FUNCTION_BLOCK FeedReactorLogic (* CAT Function Block Type *)
  (* Standard: 61499-2 *)
  (* Version 1.0, 10/1/2026, Claude/Hidryco, Schneider Electric, Rev1 - Caminho de 3 bombas reescrito (FeedReactor3PsBasic Rev1): mesmo funcionamento da Water Discharge; PID unico (PIDISc.RunPID1/Setpoint1); velocidade unica via SpeedGate (reenvio 1 s); rodizio por horimetro (FB_OPD); velocidade real (FB_SPEED); pH/condutividade pelos alarmes L/H (narrativa); reatores recebem disponibilidade/rodando de qualquer bomba; removidos SpeedSp1-3, InfluentCofiguration, INT2BOOL e WaitingTime (caminho de 1 bomba nao usado) *)
  PACKAGE SE.Nereda;
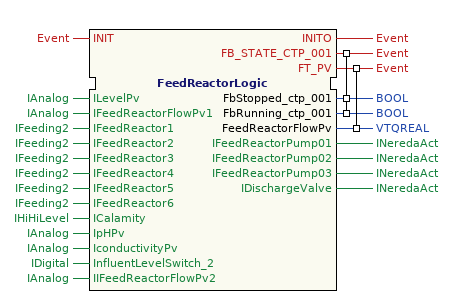
  EVENT_INPUT
    INIT;
  END_EVENT
  EVENT_OUTPUT
    INITO;
    FB_STATE_CTP_001 WITH FbStopped_ctp_001, FbRunning_ctp_001;
    FT_PV WITH FeedReactorFlowPv; (* Request for new value and limits *)
  END_EVENT
  VAR_OUTPUT
    FbStopped_ctp_001 : BOOL;
    FbRunning_ctp_001 : BOOL;
    FeedReactorFlowPv : VTQREAL; (* Vtq value *)
  END_VAR
  SOCKETS
    ILevelPv : IAnalog;
    IFeedReactorFlowPv1 : IAnalog;
    IFeedReactor1 : IFeeding2;
    IFeedReactor2 : IFeeding2;
    IFeedReactor3 : IFeeding2;
    IFeedReactor4 : IFeeding2;
    IFeedReactor5 : IFeeding2;
    IFeedReactor6 : IFeeding2;
    ICalamity : IHiHiLevel;
    IpHPv : IAnalog;
    IconductivityPv : IAnalog;
    InfluentLevelSwitch_2 : IDigital;
  END_SOCKETS
  SOCKETS
    IIFeedReactorFlowPv2 : IAnalog; (* Process value (range considered) interface adapter *)
  END_SOCKETS
  PLUGS
    IFeedReactorPump01 : INeredaAct;
    IFeedReactorPump02 : INeredaAct;
    IFeedReactorPump03 : INeredaAct;
    IDischargeValve : INeredaAct;
  END_PLUGS
  (* 01 - FUNCTIONNAL INPUT INTERFACE *)
  (* 00 - INITIALIZATION *)
  (* 05 - LOGIC *)
  (* 06 - HMI INTERFACE *)
  (* 03 - FIELD INTERFACE *)
  (* Feed Reactor Logic (One Pump) *)
  (* 02 - FUNCTIONNAL OUTPUT INTERFACE *)
  (* Interlock *)
  (* Feed Reactor Logic (3 Pumps) *)
  (* Capacity Setpoint *)
  (* Stop Pumps Cdts : The feed to the reactor must be stopped in the following situations: • Low Low level influent buffer; • pH value influent buffer too low or too high; • conductivity influent buffer too low or too high. *)
  FBS
    IThis : FeedReactorLogic_HMI(QI := TRUE);
    FeedReactorFlowPv_Status : decodeStatus; {SET_ATTRIBUTE(Configuration.Component.HideUnusedPorts, )}
    CmdPumpSmooth : boolValueChanged;
    CmdValveSmooth : boolValueChanged;
    PID : PID;
    LowLowFlow_ctp001 : ilckCondItem(CondCause := Active1);
    LowLowFlowAlarm : AND_88A3DD8EC65DD11C; {SET_ATTRIBUTE(Configuration.GenericFBType.InterfaceParams, Runtime.Standard#CNT:=2;OUT:BOOL)}
    FeedReactor1PLogic : FeedReactor1PBasic;
    LevelPv_Status : decodeStatus;
    ForceStopPump : OR_88A3DD8EC65DD11C(IN1 := FALSE); {SET_ATTRIBUTE(Configuration.GenericFBType.InterfaceParams, Runtime.Standard#CNT:=2;OUT:BOOL)}
    RESET_BTNs : RESET_BTNs;
    LoLoFlowAlarmManager : DelayedActive(pin_4E076A4928A0DFEF := TRUE, pin_1CE054BDD0AD4DEB := T#1m);
    HighHighLevel_Calamity : ilckCondItem(CondCause := Active1);
    HighHighCalamity : OR_88A3DD8EC65DD11C; {SET_ATTRIBUTE(Configuration.GenericFBType.InterfaceParams, Runtime.Standard#CNT:=2;OUT:BOOL)}
    CmdPump : BOOL2INT;
    CmdValve : BOOL2INT;
    ResetReq : OR_1147623A96AA66A8; {SET_ATTRIBUTE(Configuration.GenericFBType.InterfaceParams, Runtime.Standard#CNT:=7;OUT:BOOL)}
    FeedPumpFbMng : FeedPumpFbReactor;
    FeedReactor3PsLogic : FeedReactor3PsBasic; {SET_ATTRIBUTE(Configuration.Component.HideUnusedPorts, )}
    CmdPump1Smooth : boolValueChanged;
    CmdPump2Smooth : boolValueChanged;
    CmdPump1 : BOOL2INT;
    CmdPump2 : BOOL2INT;
    CmdPump3Smooth : boolValueChanged;
    CmdPump3 : BOOL2INT;
    ForceStop : OR_169B00D031196E7C4; {SET_ATTRIBUTE(Configuration.GenericFBType.InterfaceParams, Runtime.Standard#CNT:=4;OUT:BOOL)}
    pH_Status : decodeStatus; {SET_ATTRIBUTE(Configuration.Component.HideUnusedPorts, )}
    conductivity_Status : decodeStatus; {SET_ATTRIBUTE(Configuration.Component.HideUnusedPorts, )}
    PIDISc : PID3_Manager;
    OR1 : OR_550FE6D62F509EB3; {SET_ATTRIBUTE(Configuration.GenericFBType.InterfaceParams, Runtime.Standard#CNT:=3;OUT:BOOL)}
    INT2BOOL1 : INT2BOOL;
    TickCycle : E_CYCLE(DT := T#1s);
    SpeedGate : E_PERMIT;
    Autotune1 : Autotune;
  END_FBS
  EVENT_CONNECTIONS
    LowLowFlowAlarm.CNF TO LowLowFlow_ctp001.REQ;
    IFeedReactorFlowPv1.REQ_STATUS TO FeedReactorFlowPv_Status.REQ;
    FeedReactorFlowPv_Status.CNF TO LowLowFlowAlarm.REQ;
    ILevelPv.REQ_STATUS TO LevelPv_Status.REQ;
    LowLowFlowAlarm.CNF TO ForceStopPump.REQ;
    OR1.CNF TO ForceStopPump.REQ;
    INIT TO IThis.DA969393F6D27920;
    IThis.A8EF0BC2917800E0 TO IThis.3D88186A4172EAF0;
    HighHighCalamity.CNF TO HighHighLevel_Calamity.REQ;
    FeedReactor1PLogic.078EA09CED294ADE TO IThis.ACDDFE951F9AC365;
    RESET_BTNs.920962203CA54948 TO IThis.B1F8118D15146EFE;
    IThis.25C5B7DA6CF97B41 TO FeedReactor1PLogic.A69A10F93A67179B;
    IThis.25C5B7DA6CF97B41 TO RESET_BTNs.AB695E9A35A20E19;
    IThis.67B3DB0A1F2CCD1E TO RESET_BTNs.AB695E9A35A20E19;
    OR1.CNF TO IFeedReactor1.5A11906EF1EE87B0;
    OR1.CNF TO IFeedReactor2.5A11906EF1EE87B0;
    OR1.CNF TO IFeedReactor3.5A11906EF1EE87B0;
    OR1.CNF TO IFeedReactor4.5A11906EF1EE87B0;
    OR1.CNF TO IFeedReactor5.5A11906EF1EE87B0;
    OR1.CNF TO IFeedReactor6.5A11906EF1EE87B0;
    OR1.CNF TO CmdPump.DD5870AA881150BB;
    IFeedReactorFlowPv1.REQ TO IFeedReactor1.7593DE3331C575B6;
    IFeedReactorFlowPv1.REQ TO IFeedReactor2.7593DE3331C575B6;
    IFeedReactorFlowPv1.REQ TO IFeedReactor3.7593DE3331C575B6;
    IFeedReactorFlowPv1.REQ TO IFeedReactor4.7593DE3331C575B6;
    IFeedReactorFlowPv1.REQ TO IFeedReactor5.7593DE3331C575B6;
    IFeedReactorFlowPv1.REQ TO IFeedReactor6.7593DE3331C575B6;
    IFeedReactorPump01.CC753684FA882790 TO IFeedReactor3.70EEE9F2AA8AC204;
    IFeedReactorPump01.CC753684FA882790 TO IFeedReactor4.70EEE9F2AA8AC204;
    IFeedReactorPump01.CC753684FA882790 TO IFeedReactor5.70EEE9F2AA8AC204;
    IFeedReactorPump01.CC753684FA882790 TO IFeedReactor6.70EEE9F2AA8AC204;
    IFeedReactor1.74BA0DB8212F2576 TO FeedReactor1PLogic.7E30127865CFE16B;
    IFeedReactor2.74BA0DB8212F2576 TO FeedReactor1PLogic.7E30127865CFE16B;
    IFeedReactor3.74BA0DB8212F2576 TO FeedReactor1PLogic.7E30127865CFE16B;
    IFeedReactor4.74BA0DB8212F2576 TO FeedReactor1PLogic.7E30127865CFE16B;
    IFeedReactor5.74BA0DB8212F2576 TO FeedReactor1PLogic.7E30127865CFE16B;
    IFeedReactor6.74BA0DB8212F2576 TO FeedReactor1PLogic.7E30127865CFE16B;
    IFeedReactor1.8D6216DA6F1D1AB3 TO FeedReactor1PLogic.595E94AC272AAE70;
    IFeedReactor2.8D6216DA6F1D1AB3 TO FeedReactor1PLogic.595E94AC272AAE70;
    IFeedReactor3.8D6216DA6F1D1AB3 TO FeedReactor1PLogic.595E94AC272AAE70;
    IFeedReactor4.8D6216DA6F1D1AB3 TO FeedReactor1PLogic.595E94AC272AAE70;
    IFeedReactor5.8D6216DA6F1D1AB3 TO FeedReactor1PLogic.595E94AC272AAE70;
    IFeedReactor6.8D6216DA6F1D1AB3 TO FeedReactor1PLogic.595E94AC272AAE70;
    IDischargeValve.9CD053F8408797ED TO FeedReactor1PLogic.FBAC3AB0F3E1774A;
    IFeedReactorPump01.9CD053F8408797ED TO FeedReactor1PLogic.8666C65DB2F34DF4;
    IFeedReactorPump01.CC753684FA882790 TO FeedReactor1PLogic.01DE5B3982687378;
    IDischargeValve.CC753684FA882790 TO FeedReactor1PLogic.EBB538FC7819A0F0;
    ForceStopPump.CNF TO FeedReactor1PLogic.4BDCB67B4FFE0D64;
    FeedReactor1PLogic.085A47BAE233EC43 TO CmdPumpSmooth.REQ;
    FeedReactor1PLogic.BA495A2CD6F37AAA TO CmdValveSmooth.REQ;
    CmdPumpSmooth.CHD TO CmdPump.DD5870AA881150BB;
    CmdValveSmooth.CHD TO CmdValve.DD5870AA881150BB;
    IThis.A8EF0BC2917800E0 TO PIDISc.INIT;
    PIDISc.CE80458C9D5EF15A TO INITO;
    LoLoFlowAlarmManager.DDA64CDC00519DA4 TO LowLowFlowAlarm.REQ;
    ICalamity.15126F43E529BB4F TO HighHighCalamity.REQ;
    CmdValve.6FC99A5BD1C38561 TO IDischargeValve.0F1CDF9A9B4A227A;
    IFeedReactorPump01.9CD053F8408797ED TO FB_STATE_CTP_001;
    IFeedReactorFlowPv1.REQ TO FT_PV;
    IThis.67B3DB0A1F2CCD1E TO ResetReq.REQ;
    IFeedReactorPump01.9CD053F8408797ED TO ResetReq.REQ;
    ResetReq.CNF TO LoLoFlowAlarmManager.C451626F7187F42D;
    IFeedReactor2.9C2DC160D0649F17 TO ResetReq.REQ;
    IFeedReactor1.9C2DC160D0649F17 TO ResetReq.REQ;
    IFeedReactor3.9C2DC160D0649F17 TO ResetReq.REQ;
    IFeedReactor4.9C2DC160D0649F17 TO ResetReq.REQ;
    IFeedReactor5.9C2DC160D0649F17 TO ResetReq.REQ;
    IFeedReactor6.9C2DC160D0649F17 TO ResetReq.REQ;
    FeedPumpFbMng.CC5621380E74A0E0 TO IFeedReactor1.03923062E780DBFC;
    FeedPumpFbMng.CC5621380E74A0E0 TO IFeedReactor2.03923062E780DBFC;
    FeedPumpFbMng.CC5621380E74A0E0 TO IFeedReactor3.03923062E780DBFC;
    FeedPumpFbMng.CC5621380E74A0E0 TO IFeedReactor4.03923062E780DBFC;
    FeedPumpFbMng.CC5621380E74A0E0 TO IFeedReactor5.03923062E780DBFC;
    FeedPumpFbMng.CC5621380E74A0E0 TO IFeedReactor6.03923062E780DBFC;
    IFeedReactor1.64A31C18B824409C TO FeedPumpFbMng.84006066E90F70DE;
    IFeedReactor2.64A31C18B824409C TO FeedPumpFbMng.84006066E90F70DE;
    IFeedReactor3.64A31C18B824409C TO FeedPumpFbMng.84006066E90F70DE;
    IFeedReactor4.64A31C18B824409C TO FeedPumpFbMng.84006066E90F70DE;
    IFeedReactor5.64A31C18B824409C TO FeedPumpFbMng.84006066E90F70DE;
    IFeedReactor6.64A31C18B824409C TO FeedPumpFbMng.84006066E90F70DE;
    IFeedReactor1.74BA0DB8212F2576 TO FeedReactor1PLogic.595E94AC272AAE70;
    IFeedReactor2.74BA0DB8212F2576 TO FeedReactor1PLogic.595E94AC272AAE70;
    IFeedReactor3.74BA0DB8212F2576 TO FeedReactor1PLogic.595E94AC272AAE70;
    IFeedReactor4.74BA0DB8212F2576 TO FeedReactor1PLogic.595E94AC272AAE70;
    IFeedReactor5.74BA0DB8212F2576 TO FeedReactor1PLogic.595E94AC272AAE70;
    IFeedReactor6.74BA0DB8212F2576 TO FeedReactor1PLogic.595E94AC272AAE70;
    CmdPump1Smooth.CHD TO CmdPump1.DD5870AA881150BB;
    CmdPump2Smooth.CHD TO CmdPump2.DD5870AA881150BB;
    CmdPump3Smooth.CHD TO CmdPump3.DD5870AA881150BB;
    CmdPump1Smooth.CNF TO CmdPump2Smooth.REQ;
    CmdPump2Smooth.CNF TO CmdPump3Smooth.REQ;
    CmdPump2.6FC99A5BD1C38561 TO IFeedReactorPump02.0F1CDF9A9B4A227A;
    CmdPump3.6FC99A5BD1C38561 TO IFeedReactorPump03.0F1CDF9A9B4A227A;
    IpHPv.REQ_STATUS TO pH_Status.REQ;
    IconductivityPv.REQ_STATUS TO conductivity_Status.REQ;
    OR1.CNF TO ForceStop.REQ;
    pH_Status.CNF TO ForceStop.REQ;
    conductivity_Status.CNF TO ForceStop.REQ;
    InfluentLevelSwitch_2.REQ TO INT2BOOL1.DD5870AA881150BB;
    INT2BOOL1.6FC99A5BD1C38561 TO OR1.REQ;
    LevelPv_Status.CNF TO OR1.REQ;
    IThis.A8EF0BC2917800E0 TO TickCycle.START;
    TickCycle.EO TO FeedReactor3PsLogic.471C3CADA717EC13;
    TickCycle.EO TO SpeedGate.EI;
    FeedReactor3PsLogic.54C5C4335FC174B1 TO SpeedGate.EI;
    SpeedGate.EO TO IFeedReactorPump01.1E00729184986247;
    IFeedReactorPump01.9CD053F8408797ED TO FeedReactor3PsLogic.8666C65DB2F34DF4;
    IFeedReactorPump01.CC753684FA882790 TO FeedReactor3PsLogic.01DE5B3982687378;
    IFeedReactorPump01.2DA8AEC15204E92D TO FeedReactor3PsLogic.168409FF111F0B5A;
    IFeedReactorPump01.F846995A4121D865 TO FeedReactor3PsLogic.5E41A10D869921BD;
    SpeedGate.EO TO IFeedReactorPump02.1E00729184986247;
    IFeedReactorPump02.9CD053F8408797ED TO FeedReactor3PsLogic.8666C65DB2F34DF4;
    IFeedReactorPump02.CC753684FA882790 TO FeedReactor3PsLogic.01DE5B3982687378;
    IFeedReactorPump02.2DA8AEC15204E92D TO FeedReactor3PsLogic.168409FF111F0B5A;
    IFeedReactorPump02.F846995A4121D865 TO FeedReactor3PsLogic.5E41A10D869921BD;
    SpeedGate.EO TO IFeedReactorPump03.1E00729184986247;
    IFeedReactorPump03.9CD053F8408797ED TO FeedReactor3PsLogic.8666C65DB2F34DF4;
    IFeedReactorPump03.CC753684FA882790 TO FeedReactor3PsLogic.01DE5B3982687378;
    IFeedReactorPump03.2DA8AEC15204E92D TO FeedReactor3PsLogic.168409FF111F0B5A;
    IFeedReactorPump03.F846995A4121D865 TO FeedReactor3PsLogic.5E41A10D869921BD;
    FeedReactor3PsLogic.085A47BAE233EC43 TO CmdPump1Smooth.REQ;
    CmdPump1.6FC99A5BD1C38561 TO IFeedReactorPump01.0F1CDF9A9B4A227A;
    IFeedReactor1.74BA0DB8212F2576 TO FeedReactor3PsLogic.7E30127865CFE16B;
    IFeedReactor1.74BA0DB8212F2576 TO FeedReactor3PsLogic.595E94AC272AAE70;
    IFeedReactor1.8D6216DA6F1D1AB3 TO FeedReactor3PsLogic.595E94AC272AAE70;
    FeedReactor3PsLogic.FCD297844523CE03 TO IFeedReactor1.70EEE9F2AA8AC204;
    IFeedReactor2.74BA0DB8212F2576 TO FeedReactor3PsLogic.7E30127865CFE16B;
    IFeedReactor2.74BA0DB8212F2576 TO FeedReactor3PsLogic.595E94AC272AAE70;
    IFeedReactor2.8D6216DA6F1D1AB3 TO FeedReactor3PsLogic.595E94AC272AAE70;
    FeedReactor3PsLogic.FCD297844523CE03 TO IFeedReactor2.70EEE9F2AA8AC204;
    FeedReactor3PsLogic.FCD297844523CE03 TO FeedPumpFbMng.84006066E90F70DE;
    ForceStop.CNF TO FeedReactor3PsLogic.4BDCB67B4FFE0D64;
    LevelPv_Status.CNF TO FeedReactor3PsLogic.4BDCB67B4FFE0D64;
    FeedReactorFlowPv_Status.CNF TO FeedReactor3PsLogic.16643588834996DE;
    IFeedReactorFlowPv1.REQ TO FeedReactor3PsLogic.16643588834996DE;
    PID.CNF TO FeedReactor3PsLogic.0510D36B485733F5;
    FeedReactor3PsLogic.1878369CED9D9897 TO PIDISc.REQ;
    IThis.B4CA49BBBE66E908 TO FeedReactor3PsLogic.6712A6C827380130;
    IThis.C0050F7CE802CE26 TO FeedReactor3PsLogic.6712A6C827380130;
    IThis.25C5B7DA6CF97B41 TO FeedReactor3PsLogic.A69A10F93A67179B;
    FeedReactor3PsLogic.50ABF706162D6E5D TO IThis.E675E5B2A8A39442;
  END_CONNECTIONS
  DATA_CONNECTIONS
    LowLowFlowAlarm.OUT TO LowLowFlow_ctp001.CondSignal;
    IFeedReactorFlowPv1.Status TO FeedReactorFlowPv_Status.Status;
    FeedReactorFlowPv_Status.LoLoAlarm TO LowLowFlowAlarm.IN2;
    ILevelPv.Status TO LevelPv_Status.Status;
    LevelPv_Status.LoLoAlarm TO ForceStopPump.IN2;
    HighHighCalamity.OUT TO HighHighLevel_Calamity.CondSignal;
    FeedReactor1PLogic.AE321536059FD861 TO IThis.B8642C11FD7EB72C;
    IThis.F8C15B6A2368EBC2 TO FeedReactor1PLogic.2AC43BA050B74406;
    IThis.F8C15B6A2368EBC2 TO RESET_BTNs.479D4538AEFD6EE1;
    IThis.78DC25A16E3E12D4 TO RESET_BTNs.26767209E3135B52;
    OR1.OUT TO IFeedReactor1.2B9DC646C4F67E84;
    OR1.OUT TO IFeedReactor2.2B9DC646C4F67E84;
    OR1.OUT TO IFeedReactor3.2B9DC646C4F67E84;
    OR1.OUT TO IFeedReactor4.2B9DC646C4F67E84;
    OR1.OUT TO IFeedReactor5.2B9DC646C4F67E84;
    OR1.OUT TO IFeedReactor6.2B9DC646C4F67E84;
    IFeedReactorFlowPv1.Value TO IFeedReactor5.E608EE3E510ADBC9;
    IFeedReactorFlowPv1.Value TO IFeedReactor6.E608EE3E510ADBC9;
    IFeedReactorFlowPv1.Value TO IFeedReactor4.E608EE3E510ADBC9;
    IFeedReactorFlowPv1.Value TO IFeedReactor3.E608EE3E510ADBC9;
    IFeedReactorFlowPv1.Value TO IFeedReactor2.E608EE3E510ADBC9;
    IFeedReactorFlowPv1.Value TO IFeedReactor1.E608EE3E510ADBC9;
    IFeedReactorPump01.8A8A07EFCDA1443C TO IFeedReactor6.B41B0731DC9AD731;
    IFeedReactorPump01.8A8A07EFCDA1443C TO IFeedReactor5.B41B0731DC9AD731;
    IFeedReactorPump01.8A8A07EFCDA1443C TO IFeedReactor4.B41B0731DC9AD731;
    IFeedReactorPump01.8A8A07EFCDA1443C TO IFeedReactor3.B41B0731DC9AD731;
    IFeedReactor1.9A80F414E2AF6B87 TO FeedReactor1PLogic.C915B42A7E29ABA7;
    IFeedReactor2.9A80F414E2AF6B87 TO FeedReactor1PLogic.C035C9DDF73934B1;
    IFeedReactor3.9A80F414E2AF6B87 TO FeedReactor1PLogic.BA46BCD3AD3C4E0E;
    IFeedReactor4.9A80F414E2AF6B87 TO FeedReactor1PLogic.05202F12A8CD5CAE;
    IFeedReactor5.9A80F414E2AF6B87 TO FeedReactor1PLogic.D190D2DBF4763077;
    IFeedReactor6.9A80F414E2AF6B87 TO FeedReactor1PLogic.B2FBAF20E404318A;
    IFeedReactor1.D7CF71AAE7A3D95C TO FeedReactor1PLogic.9A612CE135251261;
    IFeedReactor2.D7CF71AAE7A3D95C TO FeedReactor1PLogic.6A6AFEA4D9C2F12F;
    IFeedReactor3.D7CF71AAE7A3D95C TO FeedReactor1PLogic.BA7B380D995C835B;
    IFeedReactor4.D7CF71AAE7A3D95C TO FeedReactor1PLogic.4960BF82FE0F0B7B;
    IFeedReactor5.D7CF71AAE7A3D95C TO FeedReactor1PLogic.9F7DD4F97732485F;
    IFeedReactor6.D7CF71AAE7A3D95C TO FeedReactor1PLogic.A6395326F4DA6B3E;
    IDischargeValve.7F6CC7FEB9223DF3 TO FeedReactor1PLogic.BC50782C9A580B55;
    IDischargeValve.A8D6C4A1FDCCA991 TO FeedReactor1PLogic.64E818E2A01597EE;
    IFeedReactorPump01.B762734C094A7162 TO FeedReactor1PLogic.75F1E123145AA883;
    IFeedReactorPump01.D83B5BDEFA4D797C TO FeedReactor1PLogic.C81CDED0AFB96994;
    IFeedReactorPump01.8A8A07EFCDA1443C TO FeedReactor1PLogic.7CAD63DC84CC56C8;
    IDischargeValve.8A8A07EFCDA1443C TO FeedReactor1PLogic.F956BBADAA4B04D2;
    ForceStopPump.OUT TO FeedReactor1PLogic.908589CFF2BDB3A2;
    FeedReactor1PLogic.3FD15F25AD96252C TO CmdPumpSmooth.Input;
    FeedReactor1PLogic.4F7C401724742E6F TO CmdValveSmooth.Input;
    CmdPumpSmooth.Output TO CmdPump.4573FC8F228EB71D;
    CmdValveSmooth.Output TO CmdValve.4573FC8F228EB71D;
    IFeedReactorPump01.B762734C094A7162 TO LoLoFlowAlarmManager.19546B227DE05AED;
    LoLoFlowAlarmManager.614F3125208254F6 TO LowLowFlowAlarm.IN1;
    ICalamity.C818324478A2F205 TO HighHighCalamity.IN1;
    ICalamity.96B50ADF37756FFC TO HighHighCalamity.IN2;
    CmdValve.A6DEF5F9C27C1848 TO IDischargeValve.710D7FC54EE3F35A;
    IFeedReactorPump01.D83B5BDEFA4D797C TO FbStopped_ctp_001;
    IFeedReactorPump01.B762734C094A7162 TO FbRunning_ctp_001;
    IFeedReactorFlowPv1.Value TO FeedReactorFlowPv;
    IThis.78DC25A16E3E12D4 TO ResetReq.IN1;
    ResetReq.OUT TO LoLoFlowAlarmManager.45767490F5BA3A44;
    IFeedReactor1.48C5E5A256C6457A TO ResetReq.IN2;
    IFeedReactor2.48C5E5A256C6457A TO ResetReq.IN3;
    IFeedReactor3.48C5E5A256C6457A TO ResetReq.IN4;
    IFeedReactor4.48C5E5A256C6457A TO ResetReq.IN5;
    IFeedReactor5.48C5E5A256C6457A TO ResetReq.IN6;
    IFeedReactor6.48C5E5A256C6457A TO ResetReq.IN7;
    IFeedReactor1.EAF64D7B7C3D74B7 TO FeedPumpFbMng.A47857DE84192E53;
    IFeedReactor2.EAF64D7B7C3D74B7 TO FeedPumpFbMng.67F20BB911804A76;
    IFeedReactor3.EAF64D7B7C3D74B7 TO FeedPumpFbMng.2171D4E21D5999D7;
    IFeedReactor4.EAF64D7B7C3D74B7 TO FeedPumpFbMng.442639032CD3044D;
    IFeedReactor5.EAF64D7B7C3D74B7 TO FeedPumpFbMng.89DCCC68F0BF2623;
    IFeedReactor6.EAF64D7B7C3D74B7 TO FeedPumpFbMng.F6D9007AB02A48F0;
    IFeedReactor1.7208B850FC6F172F TO FeedPumpFbMng.FE64A894527B1C14;
    IFeedReactor2.7208B850FC6F172F TO FeedPumpFbMng.6F6B570D325EF0B7;
    IFeedReactor3.7208B850FC6F172F TO FeedPumpFbMng.68E81F433BC634A0;
    IFeedReactor4.7208B850FC6F172F TO FeedPumpFbMng.E715B786DDD57E55;
    IFeedReactor5.7208B850FC6F172F TO FeedPumpFbMng.B82159FC57BC806F;
    IFeedReactor6.7208B850FC6F172F TO FeedPumpFbMng.2A1140A0FE0B782C;
    FeedPumpFbMng.7BF12AA41C8D8F02 TO IFeedReactor1.78D0DDD34C9EF9F8;
    FeedPumpFbMng.873B8F2FF1732060 TO IFeedReactor1.15E0B0692568D904;
    FeedPumpFbMng.F5D9A9D1D8A6D49C TO IFeedReactor2.15E0B0692568D904;
    FeedPumpFbMng.476BB0862FB32E64 TO IFeedReactor2.78D0DDD34C9EF9F8;
    FeedPumpFbMng.0E8C2A4D9A5327F7 TO IFeedReactor3.15E0B0692568D904;
    FeedPumpFbMng.4AF9DB91981D5F44 TO IFeedReactor3.78D0DDD34C9EF9F8;
    FeedPumpFbMng.9202BC4A40F84071 TO IFeedReactor4.15E0B0692568D904;
    FeedPumpFbMng.4515138E18FC7312 TO IFeedReactor4.78D0DDD34C9EF9F8;
    FeedPumpFbMng.1EEF0FB88445858E TO IFeedReactor5.15E0B0692568D904;
    FeedPumpFbMng.7957E5DEA7A144D8 TO IFeedReactor5.78D0DDD34C9EF9F8;
    FeedPumpFbMng.2DB817AD7057465C TO IFeedReactor6.15E0B0692568D904;
    FeedPumpFbMng.2FFD011EA6FD8002 TO IFeedReactor6.78D0DDD34C9EF9F8;
    CmdPump1Smooth.Output TO CmdPump1.4573FC8F228EB71D;
    CmdPump2Smooth.Output TO CmdPump2.4573FC8F228EB71D;
    CmdPump3Smooth.Output TO CmdPump3.4573FC8F228EB71D;
    CmdPump2.A6DEF5F9C27C1848 TO IFeedReactorPump02.710D7FC54EE3F35A;
    CmdPump3.A6DEF5F9C27C1848 TO IFeedReactorPump03.710D7FC54EE3F35A;
    IpHPv.Status TO pH_Status.Status;
    IconductivityPv.Status TO conductivity_Status.Status;
    LevelPv_Status.HiAlarm TO OR1.IN3;
    LevelPv_Status.HiHiAlarm TO OR1.IN2;
    InfluentLevelSwitch_2.Value TO INT2BOOL1.4573FC8F228EB71D;
    INT2BOOL1.A6DEF5F9C27C1848 TO OR1.IN1;
    FeedReactor3PsLogic.1340A87A57F03816 TO SpeedGate.PERMIT;
    FeedReactor3PsLogic.7FEAC15974107CEB TO IFeedReactorPump01.1BC103921BBFDA0B;
    IFeedReactorPump01.B762734C094A7162 TO FeedReactor3PsLogic.75F1E123145AA883;
    IFeedReactorPump01.D83B5BDEFA4D797C TO FeedReactor3PsLogic.C81CDED0AFB96994;
    IFeedReactorPump01.8A8A07EFCDA1443C TO FeedReactor3PsLogic.7CAD63DC84CC56C8;
    IFeedReactorPump01.C7F638DBF6B860D2 TO FeedReactor3PsLogic.03EF3D42F6EC65CA;
    IFeedReactorPump01.790C5C3BA88E0AF5 TO FeedReactor3PsLogic.9DC55F3DAAADF065;
    FeedReactor3PsLogic.3FD15F25AD96252C TO CmdPump1Smooth.Input;
    FeedReactor3PsLogic.7FEAC15974107CEB TO IFeedReactorPump02.1BC103921BBFDA0B;
    IFeedReactorPump02.B762734C094A7162 TO FeedReactor3PsLogic.EF60AF9AE01D1F40;
    IFeedReactorPump02.D83B5BDEFA4D797C TO FeedReactor3PsLogic.C1D7913723C9B3B7;
    IFeedReactorPump02.8A8A07EFCDA1443C TO FeedReactor3PsLogic.79CFF63624562F1A;
    IFeedReactorPump02.C7F638DBF6B860D2 TO FeedReactor3PsLogic.C12D87A372A0D4A1;
    IFeedReactorPump02.790C5C3BA88E0AF5 TO FeedReactor3PsLogic.64DEC646EA2296EC;
    FeedReactor3PsLogic.A51371F050C5DBE4 TO CmdPump2Smooth.Input;
    FeedReactor3PsLogic.7FEAC15974107CEB TO IFeedReactorPump03.1BC103921BBFDA0B;
    IFeedReactorPump03.B762734C094A7162 TO FeedReactor3PsLogic.AF6EDB8954CC95C9;
    IFeedReactorPump03.D83B5BDEFA4D797C TO FeedReactor3PsLogic.738AC9821F5B7683;
    IFeedReactorPump03.8A8A07EFCDA1443C TO FeedReactor3PsLogic.A8A9D7088A797CD2;
    IFeedReactorPump03.C7F638DBF6B860D2 TO FeedReactor3PsLogic.C401C148A7F20261;
    IFeedReactorPump03.790C5C3BA88E0AF5 TO FeedReactor3PsLogic.375265FC6460F988;
    FeedReactor3PsLogic.FFF29CFFBE485BA1 TO CmdPump3Smooth.Input;
    CmdPump1.A6DEF5F9C27C1848 TO IFeedReactorPump01.710D7FC54EE3F35A;
    IFeedReactor1.9A80F414E2AF6B87 TO FeedReactor3PsLogic.C915B42A7E29ABA7;
    IFeedReactor1.D7CF71AAE7A3D95C TO FeedReactor3PsLogic.9A612CE135251261;
    FeedReactor3PsLogic.06C907D918F5800E TO IFeedReactor1.B41B0731DC9AD731;
    IFeedReactor2.9A80F414E2AF6B87 TO FeedReactor3PsLogic.C035C9DDF73934B1;
    IFeedReactor2.D7CF71AAE7A3D95C TO FeedReactor3PsLogic.6A6AFEA4D9C2F12F;
    FeedReactor3PsLogic.06C907D918F5800E TO IFeedReactor2.B41B0731DC9AD731;
    FeedReactor3PsLogic.CFD70CC123F161E1 TO FeedPumpFbMng.A9764C308507B315;
    FeedReactor3PsLogic.F96B276460D1FCF4 TO FeedPumpFbMng.D91134A97D850EFE;
    pH_Status.LoAlarm TO ForceStop.IN1;
    pH_Status.HiAlarm TO ForceStop.IN2;
    conductivity_Status.LoAlarm TO ForceStop.IN3;
    conductivity_Status.HiAlarm TO ForceStop.IN4;
    ForceStop.OUT TO FeedReactor3PsLogic.908589CFF2BDB3A2;
    LevelPv_Status.LoLoAlarm TO FeedReactor3PsLogic.3AAAF48443B1CE4B;
    FeedReactorFlowPv_Status.LoLoAlarm TO FeedReactor3PsLogic.3F61CEAC196DAFFA;
    FeedReactorFlowPv_Status.FailAlarm TO FeedReactor3PsLogic.B9FEC6B18C045039;
    IFeedReactorFlowPv1.ValueMin TO FeedReactor3PsLogic.3FF978AD45867CD1;
    IFeedReactorFlowPv1.ValueMax TO FeedReactor3PsLogic.ECEC37AAF9912DE1;
    IFeedReactorFlowPv1.Value TO FeedReactor3PsLogic.61C6CAD8A62128A0;
    PID.Out TO FeedReactor3PsLogic.BFA4DE49E102B0EA;
    FeedReactor3PsLogic.2FD2CD82AAE9F327 TO PIDISc.RunPID;
    FeedReactor3PsLogic.31751C6AC08065D4 TO PIDISc.Setpoint;
    IThis.8E376F2FCDE4F86B TO FeedReactor3PsLogic.F11ED37F50C532BF;
    IThis.434CA134D4560A87 TO FeedReactor3PsLogic.2F2AC3038FC8C5AF;
    IThis.710F885ED2D04B14 TO FeedReactor3PsLogic.C6332A6DD9CA4077;
    IThis.6E892EF3E58F17EF TO FeedReactor3PsLogic.551314EBB6B4C778;
    IThis.B983C1B2276C6513 TO FeedReactor3PsLogic.88EBC3528E8AADEC;
    IThis.10B16495C79EB6A0 TO FeedReactor3PsLogic.51791C50D7ACFF08;
    IThis.86BCFD975F27C5A1 TO FeedReactor3PsLogic.7B2EFC85E80259FF;
    IThis.84BE37C651C94844 TO FeedReactor3PsLogic.652192BCEAC4BA87;
    IThis.144045E26F155DB9 TO FeedReactor3PsLogic.72685E9CC3009F17;
    IThis.F8C15B6A2368EBC2 TO FeedReactor3PsLogic.2AC43BA050B74406;
    FeedReactor3PsLogic.AE321536059FD861 TO IThis.210B62D8902FC1C8;
    FeedReactor3PsLogic.B27176F5DCAA83B1 TO IThis.806F5B4ED22423C6;
    FeedReactor3PsLogic.0C5A6CFA96D233BF TO IThis.EC0BBB2CD187C91A;
    FeedReactor3PsLogic.D0EA1B1A2197B0B9 TO IThis.28F388AFD283E2F2;
    FeedReactor3PsLogic.1421452A4EBFDDF1 TO IThis.2A8127B03A0A8854;
    FeedReactor3PsLogic.098AFC871A3CFD13 TO IThis.2B32DD80F05C24B0;
    FeedReactor3PsLogic.7FEAC15974107CEB TO IThis.51459164C500A8B5;
    FeedReactor3PsLogic.5C59000207A0D294 TO IThis.FCEDA547C1A0F67F;
    FeedReactor3PsLogic.BAFEC99BDB64D66C TO IThis.314200F87A96EDB6;
    FeedReactor3PsLogic.C9EE069C71EFDAD1 TO IThis.43011023704B7458;
    FeedReactor3PsLogic.9CF3FEEBF2B6AA5D TO IThis.CAF7985F3BD2F0DE;
    FeedReactor3PsLogic.B895CCC55F3FE220 TO IThis.3645222F496B83FD;
    FeedReactor3PsLogic.36986729985B7CC1 TO IThis.1637435F6E67D980;
    FeedReactor3PsLogic.C0C1B0C1C3199410 TO IThis.735547827F158D38;
    FeedReactor3PsLogic.87AEC4DAAD8A9CBC TO IThis.EF2AD2FF5C1C003A;
    FeedReactor3PsLogic.A57CDF738DF830C6 TO IThis.FA967D1C25DA4746;
    FeedReactor3PsLogic.490A1F3D34268C5C TO IThis.7ABE6A93E45C19D2;
    FeedReactor3PsLogic.4620777000303A22 TO IThis.68776047DC0513BE;
    FeedReactor3PsLogic.8798015E00F9DFD9 TO IThis.CC250B469F0B0597;
  END_CONNECTIONS
  ADAPTER_CONNECTIONS
    IIFeedReactorFlowPv2 TO PID.IPv;
    LowLowFlow_ctp001.ICondChainOut TO HighHighLevel_Calamity.ICondChainIn;
    PIDISc.FACD1DD4E791A86A TO PID.ISc;
    Autotune1.IAutotune TO PID.IAutotune;
  END_CONNECTIONS
END_FUNCTION_BLOCK
